TYPE Link_REP_Ethercat :
STRUCT
	Link_IN	AT%I*:UINT;
	Link_OUT AT%Q*:UINT;
END_STRUCT
END_TYPE

(* stored: Version 1.1.0.1
   DUT Link_REP_Ethercat: Id {471e2f11-ab6f-44ea-a28d-97d425488914} *)
